% RSLogix 500 project PID.RSS, saved by version 8.30.00.16 %
PROJECT "UNTITLED"    % processor: Bul.1763 MicroLogix 1100 Series B %

PROGRAM FILES
  LAD 2 "MAIN"  3 rungs
  LAD 3 "DIO"  2 rungs
  LAD 5 "CONTROL"  15 rungs

DATA FILES
  O0 OUTPUT  4 elements
  I1 INPUT  6 elements
  S2 STATUS  66 elements
  B3 BINARY  2 elements
  T4 TIMER  1 elements
  C5 COUNTER  1 elements
  R6 CONTROL  1 elements
  N7 INTEGER  4 elements
  F8 FLOAT  5 elements

LADDER 2 "MAIN"
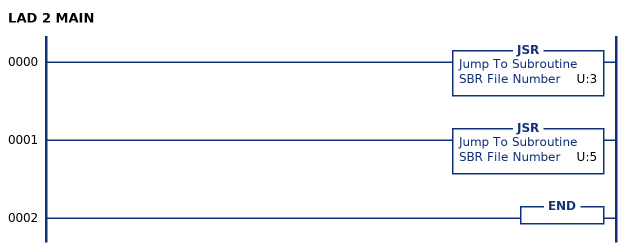
% Rung: 0 %
SOR JSR U:3 EOR
% Rung: 1 %
SOR JSR U:5 EOR
% Rung: 2 %
SOR END EOR

LADDER 3 "DIO"
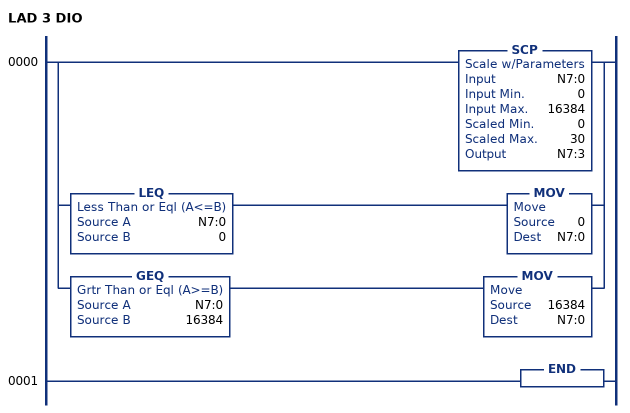
% Rung: 0 %
SOR BST SCP N7:0 0 16384 0 30 N7:3 NXB LEQ N7:0 0 MOV 0 N7:0 NXB GEQ N7:0 16384 MOV 16384 N7:0 BND EOR
% Rung: 1 %
SOR END EOR

LADDER 5 "CONTROL"
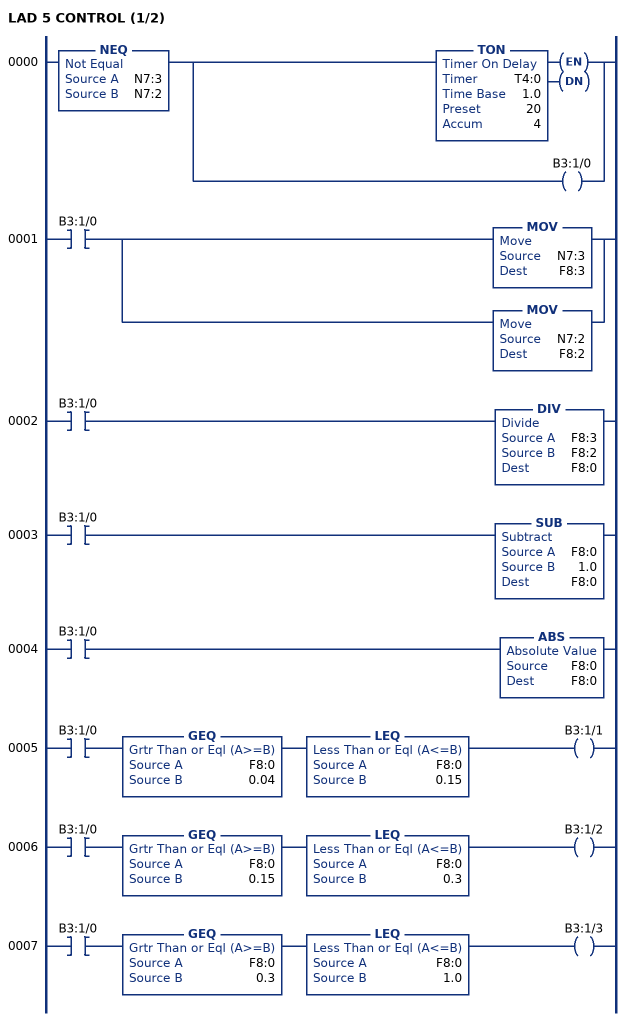
% Rung: 0 %
SOR NEQ N7:3 N7:2 BST TON T4:0 1.0 20 4 NXB OTE B3:1/0 BND EOR
% Rung: 1 %
SOR XIC B3:1/0 BST MOV N7:3 F8:3 NXB MOV N7:2 F8:2 BND EOR
% Rung: 2 %
SOR XIC B3:1/0 DIV F8:3 F8:2 F8:0 EOR
% Rung: 3 %
SOR XIC B3:1/0 SUB F8:0 1.0 F8:0 EOR
% Rung: 4 %
SOR XIC B3:1/0 ABS F8:0 F8:0 EOR
% Rung: 5 %
SOR XIC B3:1/0 GEQ F8:0 0.04 LEQ F8:0 0.15 OTE B3:1/1 EOR
% Rung: 6 %
SOR XIC B3:1/0 GEQ F8:0 0.15 LEQ F8:0 0.3 OTE B3:1/2 EOR
% Rung: 7 %
SOR XIC B3:1/0 GEQ F8:0 0.3 LEQ F8:0 1.0 OTE B3:1/3 EOR

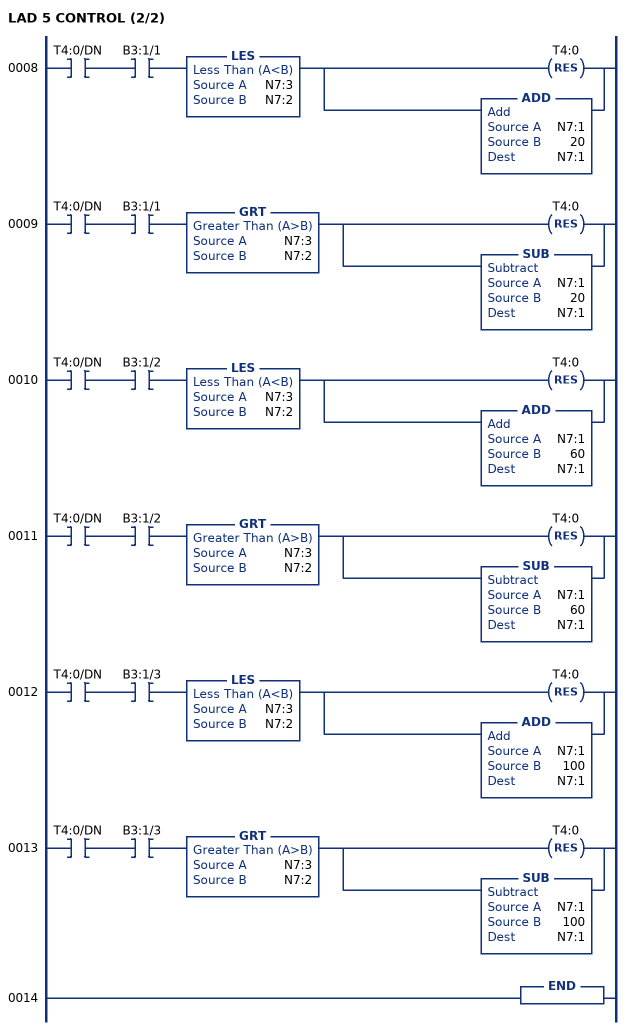
% Rung: 8 %
SOR XIC T4:0/DN XIC B3:1/1 LES N7:3 N7:2 BST RES T4:0 NXB ADD N7:1 20 N7:1 BND EOR
% Rung: 9 %
SOR XIC T4:0/DN XIC B3:1/1 GRT N7:3 N7:2 BST RES T4:0 NXB SUB N7:1 20 N7:1 BND EOR
% Rung: 10 %
SOR XIC T4:0/DN XIC B3:1/2 LES N7:3 N7:2 BST RES T4:0 NXB ADD N7:1 60 N7:1 BND EOR
% Rung: 11 %
SOR XIC T4:0/DN XIC B3:1/2 GRT N7:3 N7:2 BST RES T4:0 NXB SUB N7:1 60 N7:1 BND EOR
% Rung: 12 %
SOR XIC T4:0/DN XIC B3:1/3 LES N7:3 N7:2 BST RES T4:0 NXB ADD N7:1 100 N7:1 BND EOR
% Rung: 13 %
SOR XIC T4:0/DN XIC B3:1/3 GRT N7:3 N7:2 BST RES T4:0 NXB SUB N7:1 100 N7:1 BND EOR
% Rung: 14 %
SOR END EOR

DATA TABLE (non-zero values as saved)
DATA B3
% B3:0 % 0X0000 0X0009
DATA T4
% .PRE .ACC %
% T4:0 % 20 4
DATA N7
% N7:0 % 16384 5720 15 30
DATA F8
% F8:0 % 1 0 15 30 0
